FUNCTION_BLOCK XSLIDE_MDLL (* Transfer Slide Model with  Locally Coupled Data+Clock *)
  (* Standard: 61499-1; Classification: Model; ApplicationDomain: Simulation; Function: Bidirectional Motion *)
  (* Version 0.1, 2004-10-18, JHC, Rockwell Automation, Made LOADER an LDU_MDL. *)
  (* Version 0.0, 2004-09-27, JHC, Rockwell Automation *)
  (* Compiler header: package fb.rt.mach; import fb.rt.mva.*; import fb.rt.net.*; *)
  (* Compiler classdef: public class XSLIDE_MDLL extends FBMVCD *)
  (* Compiler Java Sun JDK 1.4.2 *)
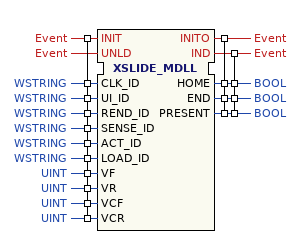
  EVENT_INPUT
    INIT WITH ACT_ID, CLK_ID, UI_ID, SENSE_ID, VF, VR, REND_ID, VCF, VCR, LOAD_ID; (* Initialize *)
    UNLD; (* Unload Workpiece *)
  END_EVENT
  EVENT_OUTPUT
    INITO WITH HOME, END, PRESENT;
    IND WITH HOME, END, PRESENT; (* Sensor Changed *)
  END_EVENT
  VAR_INPUT
    CLK_ID : WSTRING := "SIM_CLK"; (* Simulation clock channel ID *)
    UI_ID : WSTRING; (* User input channel ID from View *)
    REND_ID : WSTRING; (* Local Channel ID for Rendering Data *)
    SENSE_ID : WSTRING; (* Sensor data channel ID to Controller *)
    ACT_ID : WSTRING; (* Actuator data channel ID from Controller *)
    LOAD_ID : WSTRING; (* Workpiece loading data channel ID from Model *)
    VF : UINT; (* Forward speed in % Full Scale per CLK event *)
    VR : UINT; (* Reverse speed in %FS per CLK event *)
    VCF : UINT := 25; (* Clamp Forward speed in % Full Scale per CLK event *)
    VCR : UINT := 25; (* Clamp Reverse speed in %FS per CLK event *)
  END_VAR
  VAR_OUTPUT
    HOME : BOOL := 1; (* HOME position limit switch with hysteresis *)
    END : BOOL; (* END position limit switch with hysteresis *)
    PRESENT : BOOL; (* Workpiece Present *)
  END_VAR
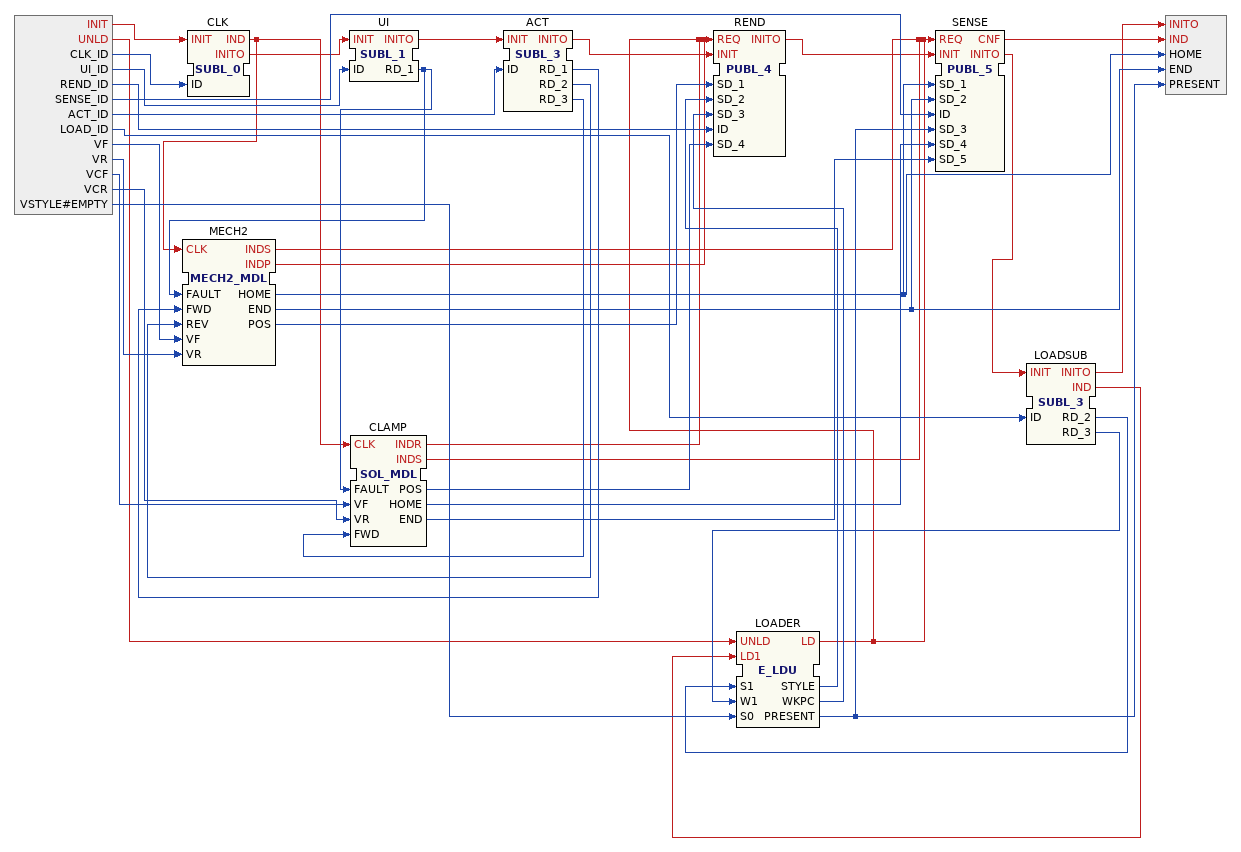
  FBS
    MECH2 : MECH2_MDL;
    UI : SUBL_1;
    CLK : SUBL_0;
    ACT : SUBL_3;
    SENSE : PUBL_5;
    REND : PUBL_4;
    LOADER : E_LDU;
    CLAMP : SOL_MDL;
    LOADSUB : SUBL_3; (* Subscriber for Load Channel *)
  END_FBS
  EVENT_CONNECTIONS
    CLK.IND TO MECH2.CLK;
    INIT TO CLK.INIT;
    MECH2.INDS TO SENSE.REQ;
    LOADER.LD TO REND.REQ;
    MECH2.INDP TO REND.REQ;
    UNLD TO LOADER.UNLD;
    LOADER.LD TO SENSE.REQ;
    SENSE.CNF TO IND;
    CLAMP.INDR TO REND.REQ;
    CLAMP.INDS TO SENSE.REQ;
    CLK.IND TO CLAMP.CLK;
    CLK.INITO TO UI.INIT;
    UI.INITO TO ACT.INIT;
    ACT.INITO TO REND.INIT;
    REND.INITO TO SENSE.INIT;
    SENSE.INITO TO LOADSUB.INIT;
    LOADSUB.INITO TO INITO;
    LOADSUB.IND TO LOADER.LD1;
  END_CONNECTIONS
  DATA_CONNECTIONS
    UI.RD_1 TO MECH2.FAULT;
    CLK_ID TO CLK.ID;
    UI_ID TO UI.ID;
    ACT_ID TO ACT.ID;
    ACT.RD_1 TO MECH2.FWD;
    ACT.RD_2 TO MECH2.REV;
    MECH2.HOME TO SENSE.SD_1;
    MECH2.END TO SENSE.SD_2;
    SENSE_ID TO SENSE.ID;
    VF TO MECH2.VF;
    VR TO MECH2.VR;
    MECH2.POS TO REND.SD_1;
    MECH2.HOME TO HOME;
    MECH2.END TO END;
    LOADER.STYLE TO REND.SD_2;
    LOADER.WKPC TO REND.SD_3;
    LOADER.PRESENT TO SENSE.SD_3;
    LOADER.PRESENT TO PRESENT;
    REND_ID TO REND.ID;
    CLAMP.POS TO REND.SD_4;
    UI.RD_1 TO CLAMP.FAULT;
    CLAMP.HOME TO SENSE.SD_4;
    CLAMP.END TO SENSE.SD_5;
    VCF TO CLAMP.VF;
    VCR TO CLAMP.VR;
    ACT.RD_3 TO CLAMP.FWD;
    LOADSUB.RD_2 TO LOADER.S1;
    LOADSUB.RD_3 TO LOADER.W1;
    VSTYLE#EMPTY TO LOADER.S0;
    LOAD_ID TO LOADSUB.ID;
  END_CONNECTIONS
END_FUNCTION_BLOCK
